(* CODESYS project Compact_DSP.project

Project tree, tasks and I/O mapping:
  Device : 3S Texas Instruments TMS320C28x DSP CPU, 3S - Smart Software Solutions GmbH, version 3.4.1.0
    application Application
      libraries: Standard, 3.4.0.0 (System)
      task MainTask (cyclic, interval t#20ms, priority 1) calls PLC_PRG
      program PLC_PRG [ST]
*)

// Device/Application/PLC_PRG
PROGRAM PLC_PRG
VAR
	A :UDINT;
END_VAR

A := A +1;

END_PROGRAM
